// TIA Portal V18 export
// export: Created 2026-06-09T02:47:52.7726546Z, ExportSetting WithDefaults, DisplayName Totally Integrated Automation Portal, DisplayVersion V18, DisplayName TIA Portal Openness, DisplayVersion V18, DisplayName TIA Portal Version Control Interface, DisplayVersion V18, DisplayName STEP 7 Professional, DisplayVersion V18, DisplayName STEP 7 Safety, DisplayVersion V18, DisplayName WinCC Professional, DisplayVersion V18
FUNCTION_BLOCK "Nalewarka"   // FB1, LAD
{ S7_Optimized_Access := 'TRUE' }
VERSION : 0.1
// stored: AutoNumber true, IsIECCheckEnabled false, IsRetainMemResEnabled false, MemoryReserve 100, SetENOAutomatically false, UDAEnableTagReadback false
   VAR
      czas_nalewarka : Time;
   END_VAR
   VAR_TEMP   // added for the SCL form of the ladder/FBD networks
      _w1 : Bool;
   END_VAR
BEGIN

REGION Network 1
   // Start przenośnika taśmowego i zapalenie się lampy sygnalizacyjnej.
   // Wyłącznik nalewarki znajduje się fizycznie na linii produkcyjnej, w jego skład wchodzi również system ryglowania. Stop natomiast w panelu HMI.
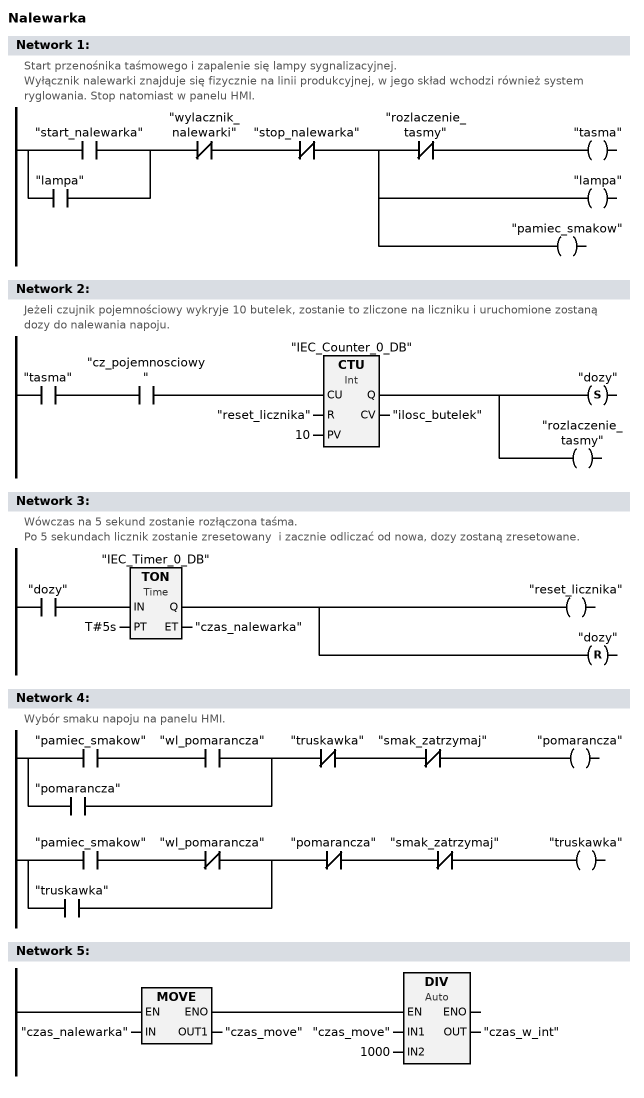
   RUNG wire#powerrail
      Contact( "start_nalewarka" )
      wire#w1
      I_Contact( "wylacznik_nalewarki" )
      I_Contact( "stop_nalewarka" )
      wire#w2
      I_Contact( "rozlaczenie_tasmy" )
      Coil( "tasma" )
   END_RUNG
   RUNG wire#powerrail
      Contact( "lampa" )
   END_RUNG wire#w1
   RUNG wire#w2
      Coil( "lampa" )
   END_RUNG
   RUNG wire#w2
      Coil( "pamiec_smakow" )
   END_RUNG
   // the same network as SCL:
   #_w1 := ("start_nalewarka" OR "lampa") AND NOT "wylacznik_nalewarki" AND NOT "stop_nalewarka";
   "tasma" := #_w1 AND NOT "rozlaczenie_tasmy";
   "lampa" := #_w1;
   "pamiec_smakow" := #_w1;
END_REGION

REGION Network 2
   // Jeżeli czujnik pojemnościowy wykryje 10 butelek, zostanie to zliczone na liczniku i uruchomione zostaną dozy do nalewania napoju.
   RUNG wire#powerrail
      Contact( "tasma" )
      Contact( "cz_pojemnosciowy" )
      { S7_Templates := "value_type := Int" } "IEC_Counter_0_DB".CTU(r := "reset_licznika", pv := 10, cv => "ilosc_butelek")
      wire#w1
      S_Coil( "dozy" )
   END_RUNG
   RUNG wire#w1
      Coil( "rozlaczenie_tasmy" )
   END_RUNG
   // the same network as SCL:
   "IEC_Counter_0_DB".CTU(CU := "tasma" AND "cz_pojemnosciowy",
                          R := "reset_licznika",
                          PV := 10,
                          CV => "ilosc_butelek");
   IF "IEC_Counter_0_DB".Q THEN "dozy" := TRUE; END_IF;
   "rozlaczenie_tasmy" := "IEC_Counter_0_DB".Q;
END_REGION

REGION Network 3
   // Wówczas na 5 sekund zostanie rozłączona taśma.
   // Po 5 sekundach licznik zostanie zresetowany  i zacznie odliczać od nowa, dozy zostaną zresetowane.
   RUNG wire#powerrail
      Contact( "dozy" )
      { S7_Templates := "time_type := Time" } "IEC_Timer_0_DB".TON(pt := T#5s, et => "czas_nalewarka")
      wire#w1
      Coil( "reset_licznika" )
   END_RUNG
   RUNG wire#w1
      R_Coil( "dozy" )
   END_RUNG
   // the same network as SCL:
   "IEC_Timer_0_DB".TON(IN := "dozy", PT := T#5s, ET => "czas_nalewarka");
   "reset_licznika" := "IEC_Timer_0_DB".Q;
   IF "IEC_Timer_0_DB".Q THEN "dozy" := FALSE; END_IF;
END_REGION

REGION Network 4
   // Wybór smaku napoju na panelu HMI.
   RUNG wire#powerrail
      Contact( "pamiec_smakow" )
      Contact( "wl_pomarancza" )
      wire#w1
      I_Contact( "truskawka" )
      I_Contact( "smak_zatrzymaj" )
      Coil( "pomarancza" )
   END_RUNG
   RUNG wire#powerrail
      Contact( "pomarancza" )
   END_RUNG wire#w1
   RUNG wire#powerrail
      Contact( "pamiec_smakow" )
      I_Contact( "wl_pomarancza" )
      wire#w2
      I_Contact( "pomarancza" )
      I_Contact( "smak_zatrzymaj" )
      Coil( "truskawka" )
   END_RUNG
   RUNG wire#powerrail
      Contact( "truskawka" )
   END_RUNG wire#w2
   // the same network as SCL:
   "pomarancza" := (("pamiec_smakow" AND "wl_pomarancza") OR "pomarancza") AND NOT "truskawka" AND NOT "smak_zatrzymaj";
   "truskawka" := (("pamiec_smakow" AND NOT "wl_pomarancza") OR "truskawka") AND NOT "pomarancza" AND NOT "smak_zatrzymaj";
END_REGION

REGION Network 5
   RUNG wire#powerrail
      Move(in := "czas_nalewarka", out1 => "czas_move")
      Div(in1 := "czas_move", in2 := 1000, out => "czas_w_int")
   END_RUNG
   // the same network as SCL:
   "czas_move" := "czas_nalewarka";
   "czas_w_int" := "czas_move" / 1000;
END_REGION
END_FUNCTION_BLOCK
